SUBAPPLICATION Uebung_034a1_Q4 (* Numeric Value Input auf PWM Ausgang *)
  (* Standard: 61499-2; Description: Copyright (c) 2023 Meisterschulen am Ostbahnhof This program and the accompanying materials are made available under the terms of the Eclipse Public License 2.0 which is available at https://www.eclipse.org/legal/epl-2.0/ SPDX-License-Identifier: EPL-2.0 *)
  (* Version 1.0, 2023-10-23, Franz Höpfinger, Meisterschulen am Ostbahnhof *)
  IMPORT Uebungen::const::UT::DefaultPool_PWM::InputNumber_PWM_Value;
  IMPORT logiBUS::io::DQ::logiBUS_DO::Output_Q4;
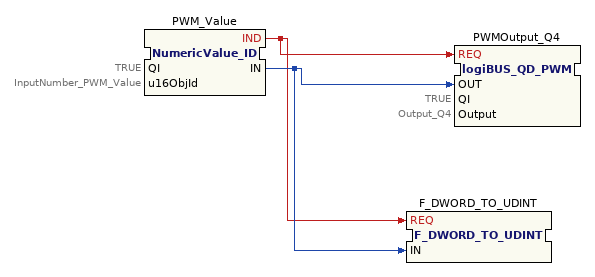
  (* ACHTUNG !! IND erscheint erst, wenn man die Numeric Value mit OK Bestätigt. nicht bei Button Druck. *)
  FBS
    F_DWORD_TO_UDINT : iec61131::conversion::F_DWORD_TO_UDINT;
    PWMOutput_Q4 : logiBUS::io::DQ::logiBUS_QD_PWM(QI := TRUE, Output := Output_Q4);
    PWM_Value : NumericValue_ID(QI := TRUE, u16ObjId := InputNumber_PWM_Value);
  END_FBS
  EVENT_CONNECTIONS
    PWM_Value.IND TO PWMOutput_Q4.REQ;
    PWM_Value.IND TO F_DWORD_TO_UDINT.REQ;
  END_CONNECTIONS
  DATA_CONNECTIONS
    PWM_Value.IN TO F_DWORD_TO_UDINT.IN;
    PWM_Value.IN TO PWMOutput_Q4.OUT;
  END_CONNECTIONS
END_SUBAPPLICATION
